Staubli VAL3: onExit.pgx

program onExit(bool x_bSave)
  local string l_sEmpty
  local num l_nResult
  local string l_sMessage
begin
//  // resetMotion
//  if !cycleStatus:bCycle
//    resetMotion()
//  endIf
//  if x_bSave
//    l_sEmpty=""
//    l_nResult=0
//    call trajType:onSave(l_sEmpty)
//    // show the message
//    call language:message(l_sMessage,-4)
//    call use:timerDialog(l_sMessage,1)
//  endIf
end
